// TIA Portal V16 export
// export: Created 2021-06-17T11:14:32.6298207Z, ExportSetting WithDefaults, DisplayName Totally Integrated Automation Portal, DisplayVersion V16 Update 4, DisplayName TIA Portal Version Control Interface, DisplayVersion V16 Update 2, DisplayName TIA Portal Openness, DisplayVersion V16 Update 4, DisplayName SINAMICS Startdrive Advanced, DisplayVersion V16 Update 5, DisplayName SINAMICS Startdrive G130, G150, S120, S150, SINAMICS MV, S210, DisplayVersion V16 Update 5, DisplayName SINAMICS Startdrive G110M, G120, G120C, G120D, G120P, G115D, DisplayVersion V16 Update 5, DisplayName STEP 7 Professional, DisplayVersion V16 Update 4, DisplayName SIMATIC Energy Suite, DisplayVersion V16 Update 4, DisplayName STEP 7 Safety, DisplayVersion V16, DisplayName WinCC Advanced / Unified PC, DisplayVersion V16 Update 4, DisplayName SIMATIC Visualization Architect, DisplayVersion V16 Update 1
DATA_BLOCK "EM_480V"   // DB9
{ S7_Optimized_Access := 'TRUE' }
VERSION : 0.1
// stored: AutoNumber true, DBAccessibleFromOPCUA true, InstanceOfName udt_EM480V_DS_142, InstanceOfType UDT, IsOnlyStoredInLoadMemory false, IsWriteProtectedInAS false
"udt_EM480V_DS_142"
   // VAR
   //    "version" { ExternalWritable := 'False'} : Byte;
   //    reserved { ExternalWritable := 'False'} : Byte;
   //    uL1N { ExternalWritable := 'False'} : Real;
   //    uL2N { ExternalWritable := 'False'} : Real;
   //    uL3N { ExternalWritable := 'False'} : Real;
   //    uL12 { ExternalWritable := 'False'} : Real;
   //    uL23 { ExternalWritable := 'False'} : Real;
   //    uL31 { ExternalWritable := 'False'} : Real;
   //    iL1 { ExternalWritable := 'False'} : Real;
   //    iL2 { ExternalWritable := 'False'} : Real;
   //    iL3 { ExternalWritable := 'False'} : Real;
   //    pfL1 { ExternalWritable := 'False'} : Real;
   //    pfL2 { ExternalWritable := 'False'} : Real;
   //    pfL3 { ExternalWritable := 'False'} : Real;
   //    pfTotal { ExternalWritable := 'False'} : Real;
   //    frequency { ExternalWritable := 'False'} : Real;
   //    amplitudeUnbalanceForVoltage { ExternalWritable := 'False'} : Real;
   //    amplitudeUnbalanceForCurrent { ExternalWritable := 'False'} : Real;
   //    sL1 { ExternalWritable := 'False'} : Real;
   //    sL2 { ExternalWritable := 'False'} : Real;
   //    sL3 { ExternalWritable := 'False'} : Real;
   //    sTotal { ExternalWritable := 'False'} : Real;
   //    qL1 { ExternalWritable := 'False'} : Real;
   //    qL2 { ExternalWritable := 'False'} : Real;
   //    qL3 { ExternalWritable := 'False'} : Real;
   //    qTotal { ExternalWritable := 'False'} : Real;
   //    pL1 { ExternalWritable := 'False'} : Real;
   //    pL2 { ExternalWritable := 'False'} : Real;
   //    pL3 { ExternalWritable := 'False'} : Real;
   //    pTotal { ExternalWritable := 'False'} : Real;
   //    phaseAngleL1 { ExternalWritable := 'False'} : Real;
   //    phaseAngleL2 { ExternalWritable := 'False'} : Real;
   //    phaseAngleL3 { ExternalWritable := 'False'} : Real;
   //    appEnTotal { ExternalWritable := 'False'} : Real;
   //    reactEnTotal { ExternalWritable := 'False'} : Real;
   //    actEnTotal { ExternalWritable := 'False'} : Real;
   //    reactEnInflow { ExternalWritable := 'False'} : Real;
   //    reactEnOutflow { ExternalWritable := 'False'} : Real;
   //    actEnInflow { ExternalWritable := 'False'} : Real;
   //    actEnOutflow { ExternalWritable := 'False'} : Real;
   //    appEnTotalLR { ExternalWritable := 'False'} : LReal;
   //    reactEnTotalLR { ExternalWritable := 'False'} : LReal;
   //    actEnTotalLR { ExternalWritable := 'False'} : LReal;
   //    reactEnInflowLR { ExternalWritable := 'False'} : LReal;
   //    reactEnOutflowLR { ExternalWritable := 'False'} : LReal;
   //    actEnInflowLR { ExternalWritable := 'False'} : LReal;
   //    actEnOutflowLR { ExternalWritable := 'False'} : LReal;
   //    iNeutral { ExternalWritable := 'False'} : Real;
   // END_VAR
BEGIN
END_DATA_BLOCK
